PROGRAM System
VAR

	
	Always_ON					:	BOOL	:=TRUE;	//상시ON
	Always_OFF					:	BOOL	:=FALSE;//상시OFF

	TON_ON  					: 	TON		; 		// 0.1초 ON 타이머 인스턴스
    TON_OFF 					:	TON		; 		// 0.1초 OFF 타이머 인스턴스
	TON2_ON  					: 	TON		; 		// 1초 ON 타이머 인스턴스
    TON2_OFF 					:	TON		;		 // 1초 OFF 타이머 인스턴스
	
	IO_Test						:	BOOL	;
	Lamp_Test_Green				:	BOOL	;
	Lamp_Test_Yellow			:	BOOL	;
	Lamp_Test_Red				:	BOOL	;
	Lamp_Test_Buzzer			:	BOOL	;
	Manual_Ready : BOOL;
	
	Buzzer						:	BOOL	;
	
	Moving_Motor_Wait_Position: BOOL;
	TEST02: INT;
	TEST06: BOOL;
	Axis02_Power_ON: TON;
	Axis03_Power_ON: TON;
	Axis04_Power_ON: TON;
END_VAR
VAR // added by the converter: edge detectors and wires of the graphical bodies
    _w1 : BOOL;
    _rt1, _rt2, _rt3, _rt4, _rt5, _rt6, _rt7 : R_TRIG;
    _ft1, _ft2 : F_TRIG;
END_VAR

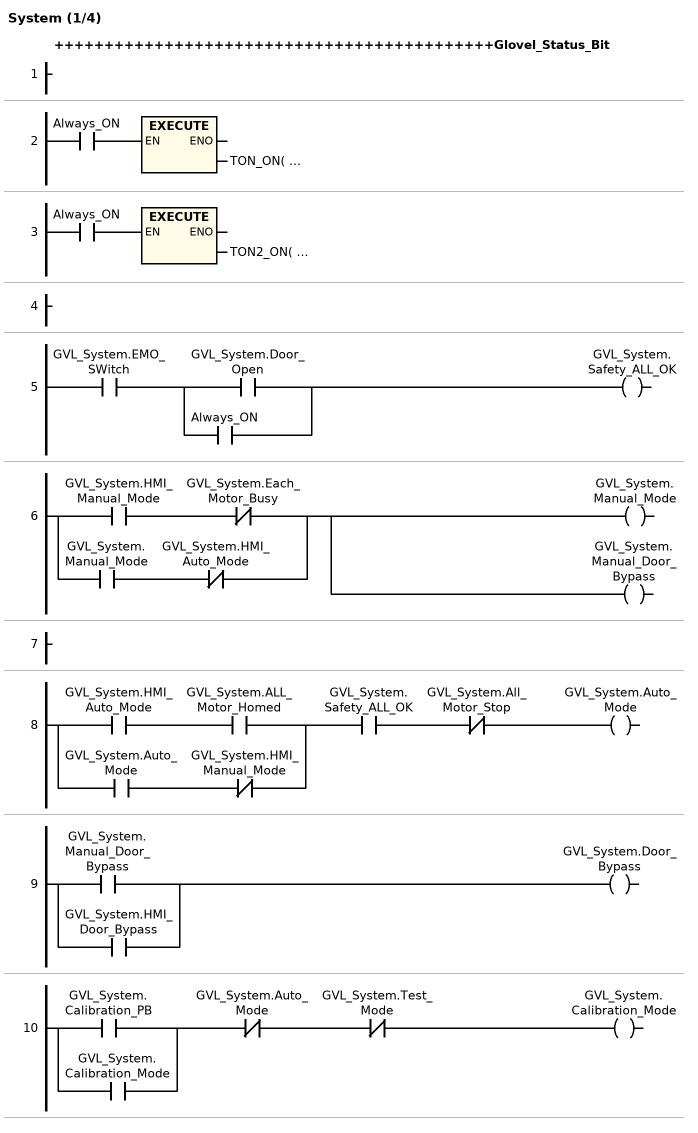
// NETWORK 1: ++++++++++++++++++++++++++++++++++++++++++++Glovel_Status_Bit

// NETWORK 2
IF Always_ON THEN
    TON_ON(
        IN := Always_ON AND NOT TON_OFF.Q,
        PT := T#100ms,
        Q  => 
    );
    
    TON_OFF(
        IN := Always_ON AND TON_ON.Q, 
        PT := T#100ms,
        Q  => 
    );
    
    GVL_System.Pulse_100ms := TON_OFF.IN;
END_IF

// NETWORK 3
IF Always_ON THEN
    TON2_ON(
        IN := Always_ON AND NOT TON2_OFF.Q,
        PT := T#1S,
        Q  => 
    );
    
    TON2_OFF(
        IN := Always_ON AND TON2_ON.Q,
        PT := T#1S,
        Q  => 
    );
    
    GVL_System.Pulse_1S := TON2_OFF.IN;
END_IF

// NETWORK 4

// NETWORK 5
GVL_System.Safety_ALL_OK := GVL_System.EMO_SWitch AND (GVL_System.Door_Open OR Always_ON);

// NETWORK 6
_w1 := GVL_System.HMI_Manual_Mode AND NOT GVL_System.Each_Motor_Busy OR GVL_System.Manual_Mode AND NOT GVL_System.HMI_Auto_Mode;
GVL_System.Manual_Mode := _w1;
GVL_System.Manual_Door_Bypass := _w1;

// NETWORK 7

// NETWORK 8
GVL_System.Auto_Mode := (GVL_System.HMI_Auto_Mode AND GVL_System.ALL_Motor_Homed OR GVL_System.Auto_Mode AND NOT GVL_System.HMI_Manual_Mode) AND GVL_System.Safety_ALL_OK AND NOT GVL_System.All_Motor_Stop;

// NETWORK 9
GVL_System.Door_Bypass := GVL_System.Manual_Door_Bypass OR GVL_System.HMI_Door_Bypass;

// NETWORK 10
GVL_System.Calibration_Mode := (GVL_System.Calibration_PB OR GVL_System.Calibration_Mode) AND NOT GVL_System.Auto_Mode AND NOT GVL_System.Test_Mode;

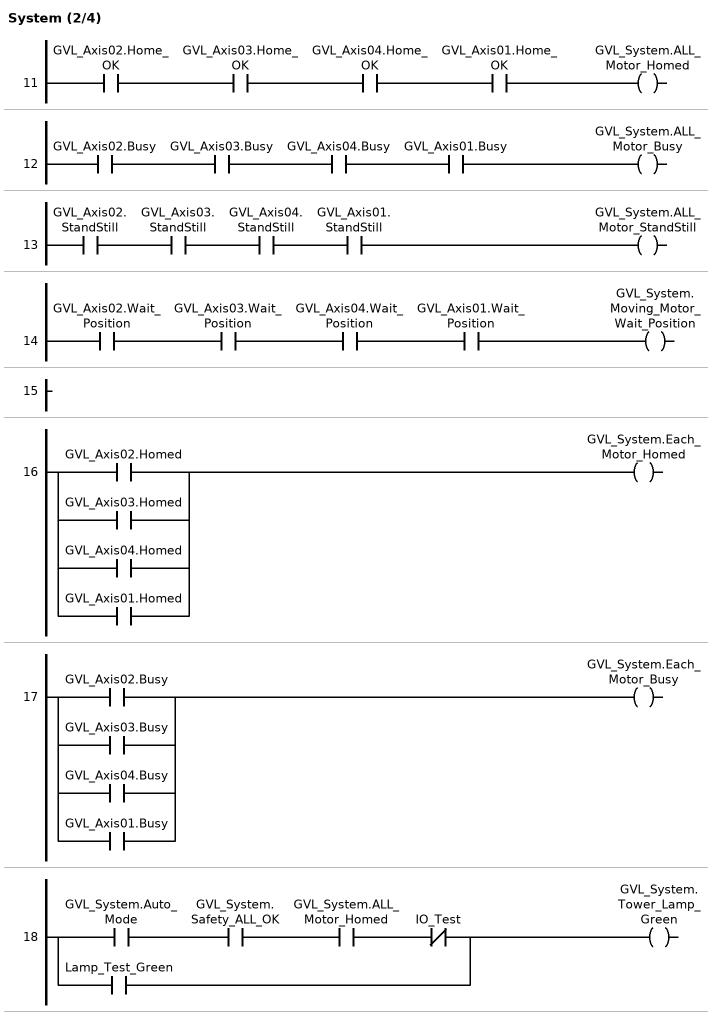
// NETWORK 11
GVL_System.ALL_Motor_Homed := GVL_Axis02.Home_OK AND GVL_Axis03.Home_OK AND GVL_Axis04.Home_OK AND GVL_Axis01.Home_OK;

// NETWORK 12
GVL_System.ALL_Motor_Busy := GVL_Axis02.Busy AND GVL_Axis03.Busy AND GVL_Axis04.Busy AND GVL_Axis01.Busy;

// NETWORK 13
GVL_System.ALL_Motor_StandStill := GVL_Axis02.StandStill AND GVL_Axis03.StandStill AND GVL_Axis04.StandStill AND GVL_Axis01.StandStill;

// NETWORK 14
GVL_System.Moving_Motor_Wait_Position := GVL_Axis02.Wait_Position AND GVL_Axis03.Wait_Position AND GVL_Axis04.Wait_Position AND GVL_Axis01.Wait_Position;

// NETWORK 15

// NETWORK 16
GVL_System.Each_Motor_Homed := GVL_Axis02.Homed OR GVL_Axis03.Homed OR GVL_Axis04.Homed OR GVL_Axis01.Homed;

// NETWORK 17
GVL_System.Each_Motor_Busy := GVL_Axis02.Busy OR GVL_Axis03.Busy OR GVL_Axis04.Busy OR GVL_Axis01.Busy;

// NETWORK 18
GVL_System.Tower_Lamp_Green := GVL_System.Auto_Mode AND GVL_System.Safety_ALL_OK AND GVL_System.ALL_Motor_Homed AND NOT IO_Test OR Lamp_Test_Green;

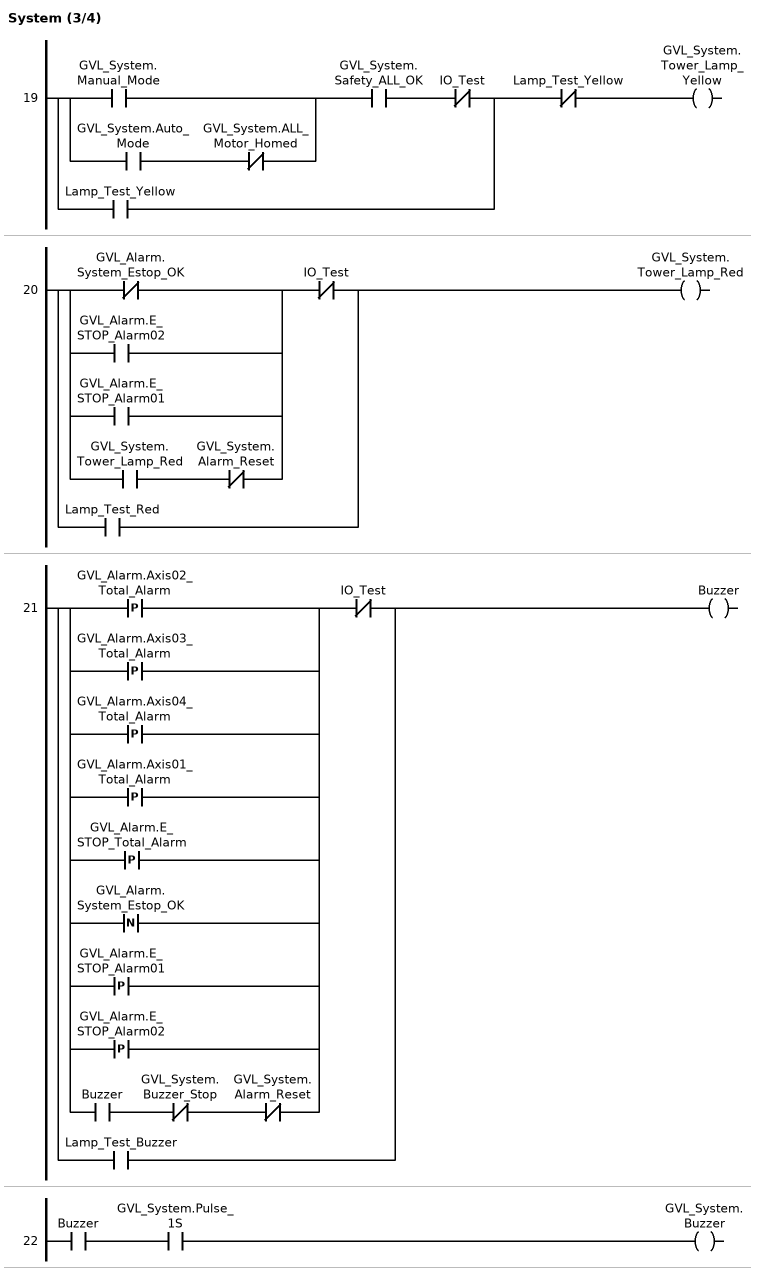
// NETWORK 19
GVL_System.Tower_Lamp_Yellow := ((GVL_System.Manual_Mode OR GVL_System.Auto_Mode AND NOT GVL_System.ALL_Motor_Homed) AND GVL_System.Safety_ALL_OK AND NOT IO_Test OR Lamp_Test_Yellow) AND NOT Lamp_Test_Yellow;

// NETWORK 20
GVL_System.Tower_Lamp_Red := (NOT GVL_Alarm.System_Estop_OK OR GVL_Alarm.E_STOP_Alarm02 OR GVL_Alarm.E_STOP_Alarm01 OR GVL_System.Tower_Lamp_Red AND NOT GVL_System.Alarm_Reset) AND NOT IO_Test OR Lamp_Test_Red;

// NETWORK 21
_rt1(CLK := GVL_Alarm.Axis02_Total_Alarm);
_rt2(CLK := GVL_Alarm.Axis03_Total_Alarm);
_rt3(CLK := GVL_Alarm.Axis04_Total_Alarm);
_rt4(CLK := GVL_Alarm.Axis01_Total_Alarm);
_rt5(CLK := GVL_Alarm.E_STOP_Total_Alarm);
_ft1(CLK := GVL_Alarm.System_Estop_OK);
_rt6(CLK := GVL_Alarm.E_STOP_Alarm01);
_rt7(CLK := GVL_Alarm.E_STOP_Alarm02);
Buzzer := (_rt1.Q OR _rt2.Q OR _rt3.Q OR _rt4.Q OR _rt5.Q OR _ft1.Q OR _rt6.Q OR _rt7.Q OR Buzzer AND NOT GVL_System.Buzzer_Stop AND NOT GVL_System.Alarm_Reset) AND NOT IO_Test OR Lamp_Test_Buzzer;

// NETWORK 22
GVL_System.Buzzer := Buzzer AND GVL_System.Pulse_1S;

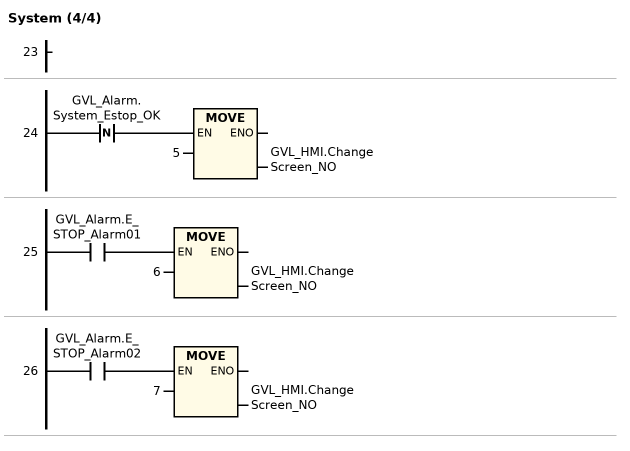
// NETWORK 23

// NETWORK 24
_ft2(CLK := GVL_Alarm.System_Estop_OK);
IF _ft2.Q THEN GVL_HMI.ChangeScreen_NO := 5; END_IF

// NETWORK 25
IF GVL_Alarm.E_STOP_Alarm01 THEN GVL_HMI.ChangeScreen_NO := 6; END_IF

// NETWORK 26
IF GVL_Alarm.E_STOP_Alarm02 THEN GVL_HMI.ChangeScreen_NO := 7; END_IF

END_PROGRAM

(* stored: Version 1.1.0.1, ProductVersion 3.1.4024.15
   POU System: Id {003f6918-e202-45f7-9f35-d63b006dbbff}, SpecialFunc None *)
